FUNCTION F_Temperature : REAL
VAR_INPUT
	Input																: INT;
	Offset																: REAL;
END_VAR
VAR
END_VAR

// F_Temperature
// Rev 1.0 - December 28, 2023

F_Temperature															:= INT_TO_REAL(Input) / 10.0 + Offset;

END_FUNCTION

(* stored: Version 1.1.0.1, ProductVersion 3.1.4024.12
   POU F_Temperature: Id {3b47d352-29a8-4ff9-a38b-2ecfd68dd430}, SpecialFunc None *)
